// TIA Portal V18 export
// export: Created 2025-12-01T17:51:27.2312606Z, ExportSetting None, DisplayName Totally Integrated Automation Portal, DisplayVersion V18 Update 5, DisplayName TIA Portal Openness, DisplayVersion V18 Update 5, DisplayName TIA Portal Teamcenter Gateway, DisplayVersion V18, DisplayName TIA Portal Version Control Interface, DisplayVersion V18, DisplayName STEP 7 Professional, DisplayVersion V18 Update 5, DisplayName STEP 7 Safety, DisplayVersion V18, DisplayName WinCC Professional, DisplayVersion V18 Update 5
DATA_BLOCK "DT-Chars_DB"   // DB2360
// stored: AutoNumber false, InstanceOfName DT-Chars, InstanceOfType FB
"DT-Chars"
   // VAR_INPUT
   //    YEAR : Int;
   //    MONTH : Int;
   //    DAY : Int;
   //    HH : Int;
   //    MM : Int;
   //    SS : Int;
   // END_VAR
   // VAR_OUTPUT
   //    Year_Byte1 : Char;
   //    Year_Byte2 : Char;
   //    Month_Byte1 : Char;
   //    Month_Byte2 : Char;
   //    Days_Byte1 : Char;
   //    Days_Byte2 : Char;
   //    HH_Byte1 : Char;
   //    HH_Byte2 : Char;
   //    MM_Byte1 : Char;
   //    MM_Byte2 : Char;
   //    SS_Byte1 : Char;
   //    SS_Byte2 : Char;
   //    CalculateDays_Byte1 : Char;
   //    CalculateDays_Byte2 : Char;
   //    CalculateDays_Byte3 : Char;
   //    Error_Code : Int;
   //    Year_Byte3 : String[1];
   //    Year_Byte4 : String[1];
   //    Month_Byte3 : String[1];
   //    Month_Byte4 : String[1];
   //    Days_Byte3 : String[1];
   //    Days_Byte4 : String[1];
   //    HH_Byte3 : String[1];
   //    HH_Byte4 : String[1];
   //    MM_Byte3 : String[1];
   //    MM_Byte4 : String[1];
   //    SS_Byte3 : String[1];
   //    SS_Byte4 : String[1];
   //    CalculateDays_Byte4 : String[1];
   //    CalculateDays_Byte5 : String[1];
   //    CalculateDays_Byte6 : String[1];
   //    OTimeStr : String[20];
   // END_VAR
   // VAR
   //    Sum_Days : Int;
   //    Sum_Year : Int;
   // END_VAR
BEGIN
END_DATA_BLOCK
